# EPICS substitutions: evrMrmApp/Db/evr-pmc-230.substitutions
# Record set for a PMC-EVR-230
#
# Macros:
#  EVR = Card name (same as mrmEvrSetupPCI())
#  SYS = System name (ie SR-TM)
#  D = Device name (ie EVR:Diag2)
#
# Record names have the general forms:
#  $(SYS){$(D)}Signal-SD
#  $(SYS){$(D)-SubDev}Signal-SD

file "evrbase.db"
{pattern
{P, OBJ, EVNT1HZ}
{"$(SYS){$(D)}", $(EVR), 125}
}

file "databuftx.db"
{pattern
{P, OBJ, PROTO}
{"$(SYS){$(D)}", "$(EVR):BUFTX", 1}
}

file "databuftxCtrl.db"
{pattern
{P, OBJ}
{"$(SYS){$(D)}", "$(EVR):BUFTX"}
}

file "mrmevrbufrx.db"
{pattern
{P, OBJ, PROTO}
{"$(SYS){$(D)}", $(EVR):BUFRX, 0xff00}
}

file "sfp.db"
{
{P="$(SYS){$(D)-SFP}", OBJ="$(EVR):SFP"}
}

file "evrmap.db"
{pattern
{NAME, OBJ, func, EVT}
{"$(SYS){$(D)}Evt:Blink0-SP", "$(EVR)", Blink, 15}
{"$(SYS){$(D)}Evt:Blink1-SP", "$(EVR)", Blink, 0}
}

file "evrevent.db"
{pattern
{EN, OBJ, CODE, EVNT}
{"$(SYS){$(D)}1hz",  "$(EVR)", 0x7d, 125}
{"$(SYS){$(D)}EvtA", "$(EVR)", 10, 10}
{"$(SYS){$(D)}EvtB", "$(EVR)", 11, 11}
{"$(SYS){$(D)}EvtC", "$(EVR)", 12, 12}
{"$(SYS){$(D)}EvtD", "$(EVR)", 13, 13}
{"$(SYS){$(D)}EvtE", "$(EVR)", 14, 14}
{"$(SYS){$(D)}EvtF", "$(EVR)", 15, 15}
{"$(SYS){$(D)}EvtG", "$(EVR)", 16, 16}
{"$(SYS){$(D)}EvtH", "$(EVR)", 17, 17}
}

file "evrscale.db"
{pattern
{IDX, P, SN, OBJ, MAX}
{0, "$(SYS){$(D)}", "$(SYS){$(D)-PS:$(IDX)}", "$(EVR):PS$(IDX)", "0xffff"}
{1, "$(SYS){$(D)}", "$(SYS){$(D)-PS:$(IDX)}", "$(EVR):PS$(IDX)", "0xffff"}
{2, "$(SYS){$(D)}", "$(SYS){$(D)-PS:$(IDX)}", "$(EVR):PS$(IDX)", "0xffff"}
}

file "mrmevrout.db"
{pattern
{ON, OBJ, DESC}
{"$(SYS){$(D)-Out:FP0}", "$(EVR):FrontOut0", "OUT0 (TTL)"}
{"$(SYS){$(D)-Out:FP1}", "$(EVR):FrontOut1", "OUT1 (TTL)"}
{"$(SYS){$(D)-Out:FP2}", "$(EVR):FrontOut2", "OUT2 (TTL)"}
}

# Pulse generators w/o a prescaler set NOPS=1
file "evrpulser.db"
{pattern
{PID, P, PN, OBJ, DMAX, WMAX, PMAX, NOPS}
{0, "$(SYS){$(D)}", "$(SYS){$(D)-DlyGen:$(PID)}", "$(EVR):Pul$(PID)", "0xffffff", "0xffff", "0xff", 0}
{1, "$(SYS){$(D)}", "$(SYS){$(D)-DlyGen:$(PID)}", "$(EVR):Pul$(PID)", "0xffffff", "0xffff", "0xff", 0}
{2, "$(SYS){$(D)}", "$(SYS){$(D)-DlyGen:$(PID)}", "$(EVR):Pul$(PID)", "0xffffff", "0xffff", "0xff", 0}
{3, "$(SYS){$(D)}", "$(SYS){$(D)-DlyGen:$(PID)}", "$(EVR):Pul$(PID)", "0xffffff", "0xffff", "0xff", 0}
{4, "$(SYS){$(D)}", "$(SYS){$(D)-DlyGen:$(PID)}", "$(EVR):Pul$(PID)", "0xffffff", "0xffff", "1", 1}
{5, "$(SYS){$(D)}", "$(SYS){$(D)-DlyGen:$(PID)}", "$(EVR):Pul$(PID)", "0xffffff", "0xffff", "1", 1}
{6, "$(SYS){$(D)}", "$(SYS){$(D)-DlyGen:$(PID)}", "$(EVR):Pul$(PID)", "0xffffff", "0xffff", "1", 1}
{7, "$(SYS){$(D)}", "$(SYS){$(D)-DlyGen:$(PID)}", "$(EVR):Pul$(PID)", "0xffffff", "0xffff", "1", 1}
{8, "$(SYS){$(D)}", "$(SYS){$(D)-DlyGen:$(PID)}", "$(EVR):Pul$(PID)", "0xffffff", "0xffff", "1", 1}
{9, "$(SYS){$(D)}", "$(SYS){$(D)-DlyGen:$(PID)}", "$(EVR):Pul$(PID)", "0xffffff", "0xffff", "1", 1}
}

# Default to 3 possible trigger mappings per pulser
file "evrpulsermap.db"
{pattern
{PID, NAME, OBJ, F, EVT}
{0, "$(SYS){$(D)-DlyGen:$(PID)}Evt:Trig0-SP", "$(EVR):Pul$(PID)", Trig, 0}
{0, "$(SYS){$(D)-DlyGen:$(PID)}Evt:Trig1-SP", "$(EVR):Pul$(PID)", Trig, 0}
{0, "$(SYS){$(D)-DlyGen:$(PID)}Evt:Trig2-SP", "$(EVR):Pul$(PID)", Trig, 0}
{1, "$(SYS){$(D)-DlyGen:$(PID)}Evt:Trig0-SP", "$(EVR):Pul$(PID)", Trig, 0}
{1, "$(SYS){$(D)-DlyGen:$(PID)}Evt:Trig1-SP", "$(EVR):Pul$(PID)", Trig, 0}
{1, "$(SYS){$(D)-DlyGen:$(PID)}Evt:Trig2-SP", "$(EVR):Pul$(PID)", Trig, 0}
{2, "$(SYS){$(D)-DlyGen:$(PID)}Evt:Trig0-SP", "$(EVR):Pul$(PID)", Trig, 0}
{2, "$(SYS){$(D)-DlyGen:$(PID)}Evt:Trig1-SP", "$(EVR):Pul$(PID)", Trig, 0}
{2, "$(SYS){$(D)-DlyGen:$(PID)}Evt:Trig2-SP", "$(EVR):Pul$(PID)", Trig, 0}
{3, "$(SYS){$(D)-DlyGen:$(PID)}Evt:Trig0-SP", "$(EVR):Pul$(PID)", Trig, 0}
{3, "$(SYS){$(D)-DlyGen:$(PID)}Evt:Trig1-SP", "$(EVR):Pul$(PID)", Trig, 0}
{3, "$(SYS){$(D)-DlyGen:$(PID)}Evt:Trig2-SP", "$(EVR):Pul$(PID)", Trig, 0}
{4, "$(SYS){$(D)-DlyGen:$(PID)}Evt:Trig0-SP", "$(EVR):Pul$(PID)", Trig, 0}
{4, "$(SYS){$(D)-DlyGen:$(PID)}Evt:Trig1-SP", "$(EVR):Pul$(PID)", Trig, 0}
{4, "$(SYS){$(D)-DlyGen:$(PID)}Evt:Trig2-SP", "$(EVR):Pul$(PID)", Trig, 0}
{5, "$(SYS){$(D)-DlyGen:$(PID)}Evt:Trig0-SP", "$(EVR):Pul$(PID)", Trig, 0}
{5, "$(SYS){$(D)-DlyGen:$(PID)}Evt:Trig1-SP", "$(EVR):Pul$(PID)", Trig, 0}
{5, "$(SYS){$(D)-DlyGen:$(PID)}Evt:Trig2-SP", "$(EVR):Pul$(PID)", Trig, 0}
{6, "$(SYS){$(D)-DlyGen:$(PID)}Evt:Trig0-SP", "$(EVR):Pul$(PID)", Trig, 0}
{6, "$(SYS){$(D)-DlyGen:$(PID)}Evt:Trig1-SP", "$(EVR):Pul$(PID)", Trig, 0}
{6, "$(SYS){$(D)-DlyGen:$(PID)}Evt:Trig2-SP", "$(EVR):Pul$(PID)", Trig, 0}
{7, "$(SYS){$(D)-DlyGen:$(PID)}Evt:Trig0-SP", "$(EVR):Pul$(PID)", Trig, 0}
{7, "$(SYS){$(D)-DlyGen:$(PID)}Evt:Trig1-SP", "$(EVR):Pul$(PID)", Trig, 0}
{7, "$(SYS){$(D)-DlyGen:$(PID)}Evt:Trig2-SP", "$(EVR):Pul$(PID)", Trig, 0}
{8, "$(SYS){$(D)-DlyGen:$(PID)}Evt:Trig0-SP", "$(EVR):Pul$(PID)", Trig, 0}
{8, "$(SYS){$(D)-DlyGen:$(PID)}Evt:Trig1-SP", "$(EVR):Pul$(PID)", Trig, 0}
{8, "$(SYS){$(D)-DlyGen:$(PID)}Evt:Trig2-SP", "$(EVR):Pul$(PID)", Trig, 0}
{9, "$(SYS){$(D)-DlyGen:$(PID)}Evt:Trig0-SP", "$(EVR):Pul$(PID)", Trig, 0}
{9, "$(SYS){$(D)-DlyGen:$(PID)}Evt:Trig1-SP", "$(EVR):Pul$(PID)", Trig, 0}
{9, "$(SYS){$(D)-DlyGen:$(PID)}Evt:Trig2-SP", "$(EVR):Pul$(PID)", Trig, 0}
}

file "evrin.db"
{pattern
{IN, OBJ, DESC}
{"$(SYS){$(D)-In:0}", "$(EVR):FPIn0", "EXT IN (TTL)"}
}
